(*
	dont we all?
*)
INTERFACE IHaveLintValue EXTENDS CNM_AbstractObject.IObject

PROPERTY value : LINT
GET
END_GET
SET
END_SET
END_PROPERTY

END_INTERFACE

(* stored: Version 1.1.0.1
   Itf IHaveLintValue: Id {3933348a-70aa-429e-9e11-3a6844995784}
   Property value: Id {97763720-a23a-4d77-800b-edce7b764b19}
   Get Get: Id {45900457-b06a-407f-8100-f0aa97ce7530}
   Set Set: Id {7736400f-f53a-4c31-ac9c-b137f29d7b9c} *)
